(* IEC 61131-3 sources: repolevel_ST_code_completion/ground_truth/repoeval_Proxy_Application/readful_result, 2 files *)

(* ---- Proxy.st ---- *)
The code fragments provided appear to be part of a structured text (ST) implementation for a Proxy design pattern in an industrial automation context, likely using IEC 61131-3 programming standards. Here's a breakdown of the functionality and relationships between the fragments:

---

### **1. Realsubject.st**
This file defines the `Realsubject` function block, which implements the `Subject_Interface`. It contains a single variable `iProp` that can be used to store and retrieve values. This function block represents the actual subject being protected by the proxy.

```st
{attribute 'enable_dynamic_creation'}
FUNCTION_BLOCK Realsubject IMPLEMENTS Subject_Interface
VAR_INPUT
END_VAR
VAR_OUTPUT
END_VAR
VAR
	// Variable to get and set values
	iProp: INT;
END_VAR
```

---

### **2. Proxy.st**
This file defines the `Proxy` function block, which also implements the `Subject_Interface`. The proxy acts as an intermediary between the client and the `Realsubject`. It includes:
- A pointer (`refToRealSubject`) to the `Realsubject` instance being protected.
- A temporary password (`iTempPassword`) entered by the client.
- A default password (`iRealPassword`) stored as a static variable.

```st
{attribute 'enable_dynamic_creation'}
FUNCTION_BLOCK Proxy IMPLEMENTS Subject_Interface
VAR_INPUT
END_VAR
VAR_OUTPUT
END_VAR
VAR
	// Pointer to store the reference to the subject being protected
	refToRealSubject : POINTER TO Realsubject;
	// Last value of password entered by the client in the visualization element
	iTempPassword : INT;
END_VAR
VAR_STAT
	// Default password value for the request to be accepted
	iRealPassword : INT := 1234;
END_VAR
```

---

### **3. Subject_Interface_Get_Method.st**
This file defines the `Get_Method`, which is part of the `Subject_Interface`. It likely retrieves the value of `iProp` from the `Realsubject`.

```st
METHOD Get_Method : INT
VAR_INPUT
END_VAR
```

---

### **4. Subject_Interface_Set_Method.st**
This file defines the `Set_Method`, which is part of the `Subject_Interface`. It sets a value (`num`) to the `iProp` variable in the `Realsubject`.

```st
METHOD Set_Method
VAR_INPUT
	// Value to be set passed as an argument
	num : INT;
END_VAR
```

---

### **5. Proxy_fb_init.st**
This file defines the `fb_init` method for the `Proxy` function block. It initializes the proxy instance with:
- A pointer to the `Realsubject` instance (`ptrToRealSubject`).
- A temporary password (`iTempPassword`) passed by the client.
- A value to be set (`iSetValue`) in case of a write request.
- A boolean (`bReadWrite`) specifying whether the request is a read or write operation.

The method also initializes the proxy's internal variables.

```st
METHOD fb_init
VAR_INPUT
	// These boolean values are required for an automatic constructor
	bInitRetains : BOOL; // TRUE: the Retain-variables are initialized (reset warm / reset cold)
	bInCopyCode : BOOL;  // TRUE: the instance will be copied to the copy-code afterward (online change)

	// Pointer to the RealSubject instance
	ptrToRealSubject : POINTER TO Realsubject;
	// Local variable to store the password passed by the client with the password of the Proxy
	iTempPassword : INT;
	// Local variable to be used in WRITE request, it is the value to be set if the request is accepted
	iSetValue : INT;
	// Boolean value that specifies if the request is a WRITE or READ request
	bReadWrite : BOOL;
END_VAR

VAR_OUTPUT
END_VAR
VAR
	// Pointer to store the reference to the subject being protected
	refToRealSubject : POINTER TO Realsubject;
	// Last value of password entered by the client in the visualization element
	iTempPassword : INT;
END_VAR
VAR_STAT
END_VAR
```

---

### **Summary**
The provided code fragments implement a Proxy design pattern where:
1. The `Realsubject` is the actual object being protected.
2. The `Proxy` acts as an intermediary, controlling access to the `Realsubject`.
3. The `Get_Method` and `Set_Method` provide interfaces for reading and writing values to the `Realsubject`.
4. The `fb_init` method initializes the `Proxy` with necessary parameters, including a pointer to the `Realsubject` and client-provided inputs.

This design pattern is useful for scenarios where access control, logging, or additional functionality is required before interacting with the actual subject.

(* ---- Proxy_1.st ---- *)
The code fragments provided appear to be part of a structured text (ST) implementation for a Proxy design pattern in an industrial automation context, likely using IEC 61131-3 programming standards. Here's a breakdown of the functionality and relationships between the fragments:

---

### **1. Realsubject.st**
This file defines the `Realsubject` function block, which implements the `Subject_Interface`. It contains a single variable `iProp` that can be used to store and retrieve values. This function block represents the actual subject being protected by the proxy.

```st
{attribute 'enable_dynamic_creation'}
FUNCTION_BLOCK Realsubject IMPLEMENTS Subject_Interface
VAR_INPUT
END_VAR
VAR_OUTPUT
END_VAR
VAR
	// Variable to get and set values
	iProp: INT;
END_VAR
```

---

### **2. Proxy.st**
This file defines the `Proxy` function block, which also implements the `Subject_Interface`. The proxy acts as an intermediary between the client and the `Realsubject`. It includes:
- A pointer (`refToRealSubject`) to the `Realsubject` instance being protected.
- A temporary password (`iTempPassword`) entered by the client.
- A default password (`iRealPassword`) stored as a static variable.

```st
{attribute 'enable_dynamic_creation'}
FUNCTION_BLOCK Proxy IMPLEMENTS Subject_Interface
VAR_INPUT
END_VAR
VAR_OUTPUT
END_VAR
VAR
	// Pointer to store the reference to the subject being protected
	refToRealSubject : POINTER TO Realsubject;
	// Last value of password entered by the client in the visualization element
	iTempPassword : INT;
END_VAR
VAR_STAT
	// Default password value for the request to be accepted
	iRealPassword : INT := 1234;
END_VAR
```

---

### **3. Subject_Interface_Get_Method.st**
This file defines the `Get_Method`, which is part of the `Subject_Interface`. It likely retrieves the value of `iProp` from the `Realsubject`.

```st
METHOD Get_Method : INT
VAR_INPUT
END_VAR
```

---

### **4. Subject_Interface_Set_Method.st**
This file defines the `Set_Method`, which is part of the `Subject_Interface`. It sets a value (`num`) to the `iProp` variable in the `Realsubject`.

```st
METHOD Set_Method
VAR_INPUT
	// Value to be set passed as an argument
	num : INT;
END_VAR
```

---

### **5. Proxy_fb_init.st**
This file defines the `fb_init` method for the `Proxy` function block. It initializes the proxy instance with:
- A pointer to the `Realsubject` instance (`ptrToRealSubject`).
- A temporary password (`iTempPassword`) passed by the client.
- A value to be set (`iSetValue`) in case of a write request.
- A boolean (`bReadWrite`) specifying whether the request is a read or write operation.

The method also initializes the proxy's internal variables.

```st
METHOD fb_init
VAR_INPUT
	// These boolean values are required for an automatic constructor
	bInitRetains : BOOL; // TRUE: the Retain-variables are initialized (reset warm / reset cold)
	bInCopyCode : BOOL;  // TRUE: the instance will be copied to the copy-code afterward (online change)

	// Pointer to the RealSubject instance
	ptrToRealSubject : POINTER TO Realsubject;
	// Local variable to store the password passed by the client with the password of the Proxy
	iTempPassword : INT;
	// Local variable to be used in WRITE request, it is the value to be set if the request is accepted
	iSetValue : INT;
	// Boolean value that specifies if the request is a WRITE or READ request
	bReadWrite : BOOL;
END_VAR

VAR_OUTPUT
END_VAR
VAR
	// Pointer to store the reference to the subject being protected
	refToRealSubject : POINTER TO Realsubject;
	// Last value of password entered by the client in the visualization element
	iTempPassword : INT;
END_VAR
VAR_STAT
END_VAR
```

---

### **Summary**
The provided code fragments implement a Proxy design pattern where:
1. The `Realsubject` is the actual object being protected.
2. The `Proxy` acts as an intermediary, controlling access to the `Realsubject`.
3. The `Get_Method` and `Set_Method` provide interfaces for reading and writing values to the `Realsubject`.
4. The `fb_init` method initializes the `Proxy` with necessary parameters, including a pointer to the `Realsubject` and client-provided inputs.

This design pattern is useful for scenarios where access control, logging, or additional functionality is required before interacting with the actual subject.
